{attribute 'qualified_only'}
{attribute 'strict'}
TYPE E_LedFunction :
(
    eUndefined := 0,
    eSteady := 1,
    eSlow := 2,
    eFast := 3
);
END_TYPE

(* stored: Version 1.1.0.1, ProductVersion 3.1.4024.11
   DUT E_LedFunction: Id {b7e49b88-88f8-4d97-8125-24afd7415e82} *)
